SUBAPPLICATION Klappen_Sitzventile (* Subapplication Type *)
  (* Standard: 61499-2 *)
  (* Version 1.0, 2023-02-11, franz *)
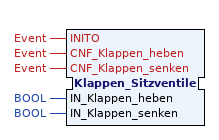
  EVENT_INPUT
    INITO;
    CNF_Klappen_heben;
    CNF_Klappen_senken;
  END_EVENT
  VAR_INPUT
    IN_Klappen_heben : BOOL;
    IN_Klappen_senken : BOOL;
  END_VAR
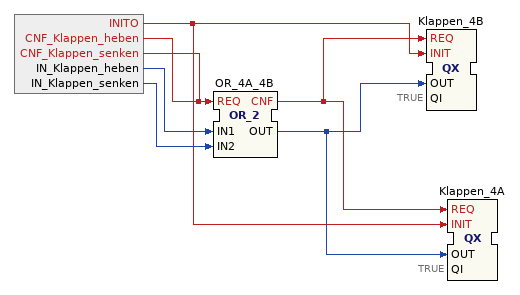
  FBS
    OR_4A_4B : OR_2; {SET_ATTRIBUTE(PinComment, IN1:Klappen_heben)} {SET_ATTRIBUTE(PinComment, IN2:Klappen_senken)}
    Klappen_4B : QX(QI := TRUE);
    Klappen_4A : QX(QI := TRUE);
  END_FBS
  EVENT_CONNECTIONS
    OR_4A_4B.CNF TO Klappen_4B.REQ;
    OR_4A_4B.CNF TO Klappen_4A.REQ;
    CNF_Klappen_heben TO OR_4A_4B.REQ;
    CNF_Klappen_senken TO OR_4A_4B.REQ;
    INITO TO Klappen_4B.INIT;
    INITO TO Klappen_4A.INIT;
  END_CONNECTIONS
  DATA_CONNECTIONS
    OR_4A_4B.OUT TO Klappen_4B.OUT;
    OR_4A_4B.OUT TO Klappen_4A.OUT;
    IN_Klappen_heben TO OR_4A_4B.IN1;
    IN_Klappen_senken TO OR_4A_4B.IN2;
  END_CONNECTIONS
END_SUBAPPLICATION
